FUNCTION_BLOCK MotVsFailures (* CAT Function Block Type *)
  (* Standard: 61499-2 *)
  (* Version 0.0, 8/5/2026, Schneider Electric, template *)
  PACKAGE SE.Nereda;
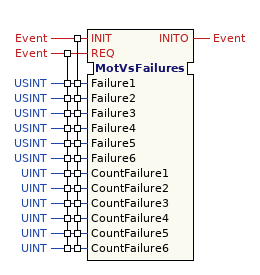
  EVENT_INPUT
    INIT WITH Failure1, Failure2, Failure3, Failure4, Failure5, Failure6, CountFailure1, CountFailure2, CountFailure3, CountFailure4, CountFailure5, CountFailure6; (* Initialization Request *)
    REQ WITH Failure1, Failure2, Failure3, Failure4, Failure5, Failure6, CountFailure1, CountFailure2, CountFailure3, CountFailure4, CountFailure5, CountFailure6;
  END_EVENT
  EVENT_OUTPUT
    INITO; (* Initialization Confirm *)
  END_EVENT
  VAR_INPUT
    Failure1 : USINT;
    Failure2 : USINT;
    Failure3 : USINT;
    Failure4 : USINT;
    Failure5 : USINT;
    Failure6 : USINT;
    CountFailure1 : UINT;
    CountFailure2 : UINT;
    CountFailure3 : UINT;
    CountFailure4 : UINT;
    CountFailure5 : UINT;
    CountFailure6 : UINT;
  END_VAR
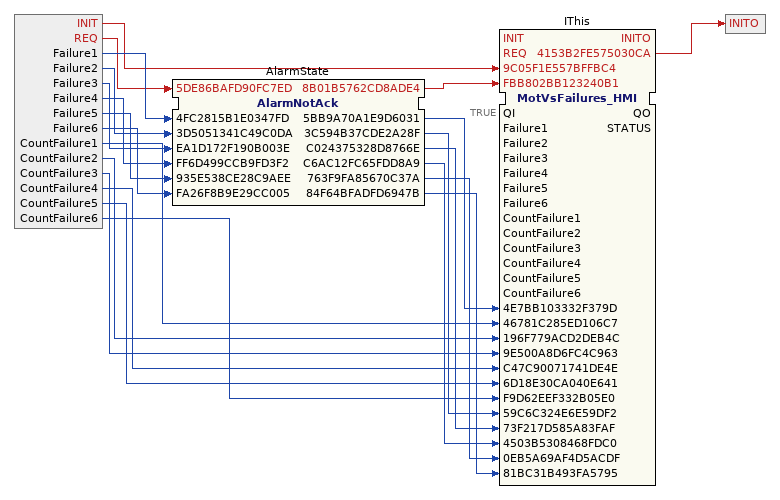
  FBS
    IThis : MotVsFailures_HMI(QI := TRUE);
    AlarmState : AlarmNotAck;
  END_FBS
  EVENT_CONNECTIONS
    REQ TO AlarmState.5DE86BAFD90FC7ED;
    INIT TO IThis.9C05F1E557BFFBC4;
    AlarmState.8B01B5762CD8ADE4 TO IThis.FBB802BB123240B1;
    IThis.4153B2FE575030CA TO INITO;
  END_CONNECTIONS
  DATA_CONNECTIONS
    Failure1 TO AlarmState.4FC2815B1E0347FD;
    AlarmState.5BB9A70A1E9D6031 TO IThis.4E7BB103332F379D;
    Failure2 TO AlarmState.3D5051341C49C0DA;
    Failure3 TO AlarmState.EA1D172F190B003E;
    Failure4 TO AlarmState.FF6D499CCB9FD3F2;
    Failure5 TO AlarmState.935E538CE28C9AEE;
    Failure6 TO AlarmState.FA26F8B9E29CC005;
    CountFailure1 TO IThis.46781C285ED106C7;
    CountFailure2 TO IThis.196F779ACD2DEB4C;
    CountFailure3 TO IThis.9E500A8D6FC4C963;
    CountFailure4 TO IThis.C47C90071741DE4E;
    CountFailure5 TO IThis.6D18E30CA040E641;
    CountFailure6 TO IThis.F9D62EEF332B05E0;
    AlarmState.3C594B37CDE2A28F TO IThis.59C6C324E6E59DF2;
    AlarmState.C024375328D8766E TO IThis.73F217D585A83FAF;
    AlarmState.C6AC12FC65FDD8A9 TO IThis.4503B5308468FDC0;
    AlarmState.763F9FA85670C37A TO IThis.0EB5A69AF4D5ACDF;
    AlarmState.84F64BFADFD6947B TO IThis.81BC31B493FA5795;
  END_CONNECTIONS
END_FUNCTION_BLOCK
